// TIA Portal V19 export
ORGANIZATION_BLOCK "Main"   // OB2011, LAD, ProgramCycle
TITLE = "Main Program Sweep (Cycle)"
// stored: AutoNumber false, IsIECCheckEnabled true, Namespace Unit.Em1, SetENOAutomatically true
   VAR_INPUT
      Initial_Call : Bool;   // Initial call of this OB
      Remanence : Bool;   // =True, if remanent data are available
   END_VAR
   VAR_TEMP
      tempIndex : Int;   // Index of EM in the array
   END_VAR
BEGIN

REGION Network 1: Call Equipment
   // Call FB CallEquipment and handover information from the unit
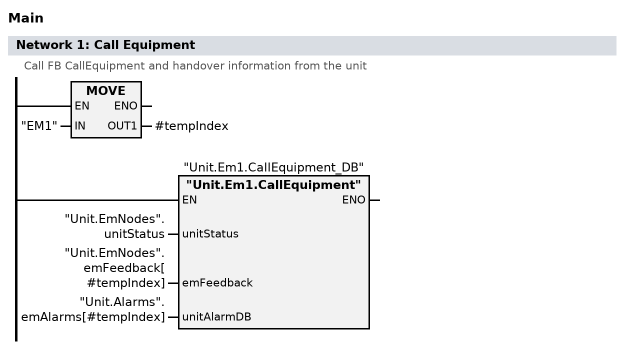
   RUNG wire#powerrail
      Move(in := "EM1", out1 => #tempIndex)
   END_RUNG
   RUNG wire#powerrail
      "Unit.Em1.CallEquipment_DB"(unitStatus := "Unit.EmNodes".unitStatus, emFeedback := "Unit.EmNodes".emFeedback[#tempIndex], unitAlarmDB := "Unit.Alarms".emAlarms[#tempIndex])
   END_RUNG
   // the same network as SCL:
   #tempIndex := "EM1";
   "Unit.Em1.CallEquipment_DB"(unitStatus := "Unit.EmNodes".unitStatus,   // "Unit.Em1.CallEquipment"
                           emFeedback := "Unit.EmNodes".emFeedback[#tempIndex],
                           unitAlarmDB := "Unit.Alarms".emAlarms[#tempIndex]);
END_REGION
END_ORGANIZATION_BLOCK
